ABB RobotStudio station: Task1_welding_1.rspag

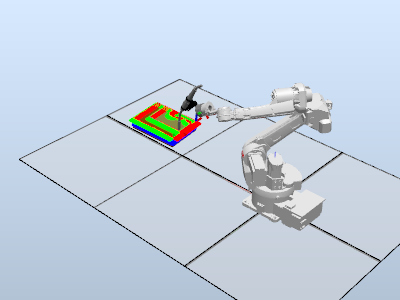
--- station ---
Station Task1_welding_1 (saved by RobotStudio 22.3.10098.0)
Controller IRB_1520ID_4kg_1.50m
  mechanical unit ROB_1: IRB1520ID_4_150__02, 6 joints, base frame (0, 0, 0) mm
Layout (positions relative to the parent item):
  - IRB1520ID_4_150__02 [mechanism, from Robots\IRB1520ID_4_150_G_02.rslib] at (0, 0, 0) mm; joint values [0.8708, -0.9702, 1.0298, -0.8942, 0.8494, 1.1291] (rad or m)
  - AW_Gun_PSF_25 [mechanism, from Tools\AW_Gun_PSF_25.rslib] at (433.02, 332.31, 841.28) mm, rotated rx 180 ry 59.43 rz -172.96 deg
  - Curve_thing [part, from Training Objects\Curve_Thing.rslib] at (696.55, 149.94, 458.64) mm, rotated rx 0 ry -5.23 rz 7.04 deg
  - Part_1 [part] at (696.55, 149.94, 458.64) mm, rotated rx 0 ry -5.23 rz 7.04 deg, size 300 x 200 x 0 mm
  - Part_2 [part] at (696.55, 149.94, 458.64) mm, rotated rx 0 ry -5.23 rz 7.04 deg, size 400 x 0 x 90 mm
Attachment: AW_Gun_PSF_25 is attached to IRB1520ID_4_150__02 / Link6

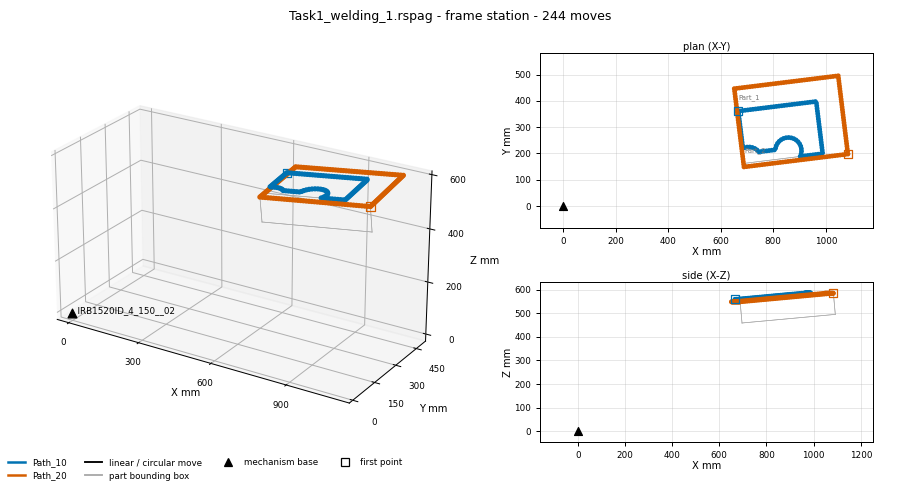
[picture p0: tool path of Task1_welding_1.rspag in frame station, 244 of 244 moves have a stored position in this frame; points joined in program order, loops and branches not executed]
--- Backups/IRB_1520ID_4kg_1.50m/RAPID/TASK1/PROGMOD/CalibData.mod ---
MODULE CalibData
	PERS tooldata AW_Gun:=[TRUE,[[119.5,0,352],[0.890213743,0,0.455543074,0]],[1,[0,0,100],[1,0,0,0],0,0,0]];
	TASK PERS wobjdata myPalletWO:=[FALSE,TRUE,"",[[688.418839009,148.925896983,548.269503166],[0.74843401,0.03415564,-0.030194721,-0.66164054]],[[0,0,0],[1,0,0,0]]];
    TASK PERS wobjdata Workobject_1:=[FALSE,TRUE,"",[[688.417832153,148.925979259,548.268984532],[0.997073299,0.002800799,-0.045502463,0.061371969]],[[0,0,0],[0,0.707106781,0.707106781,0]]];
    PROC Path_10()
        MoveJ Target_10,v1000,z100,AW_Gun\WObj:=wobj0;
        MoveL Target_20,v1000,z100,AW_Gun\WObj:=wobj0;
        MoveL Target_30,v1000,z100,AW_Gun\WObj:=wobj0;
        MoveL Target_40,v1000,z100,AW_Gun\WObj:=wobj0;
        MoveL Target_50,v1000,z100,AW_Gun\WObj:=wobj0;
        MoveL Target_60,v1000,z100,AW_Gun\WObj:=wobj0;
        MoveL Target_80,v1000,z100,AW_Gun\WObj:=wobj0;
        MoveL Target_70,v1000,z100,AW_Gun\WObj:=wobj0;
        MoveL Target_90,v1000,z100,AW_Gun\WObj:=wobj0;
        MoveL Target_100,v1000,z100,AW_Gun\WObj:=wobj0;
        MoveL Target_110,v1000,z100,AW_Gun\WObj:=wobj0;
        MoveL Target_120,v1000,z100,AW_Gun\WObj:=wobj0;
        MoveL Target_130,v1000,z100,AW_Gun\WObj:=wobj0;
        MoveL Target_140,v1000,z100,AW_Gun\WObj:=wobj0;
        MoveL Target_150,v1000,z100,AW_Gun\WObj:=wobj0;
        MoveL Target_160,v1000,z100,AW_Gun\WObj:=wobj0;
        MoveL Target_170,v1000,z100,AW_Gun\WObj:=wobj0;
        MoveL Target_180,v1000,z100,AW_Gun\WObj:=wobj0;
        MoveL Target_190,v1000,z100,AW_Gun\WObj:=wobj0;
        MoveL Target_200,v1000,z100,AW_Gun\WObj:=wobj0;
        MoveL Target_210,v1000,z100,AW_Gun\WObj:=wobj0;
        MoveL Target_220,v1000,z100,AW_Gun\WObj:=wobj0;
        MoveL Target_230,v1000,z100,AW_Gun\WObj:=wobj0;
        MoveL Target_240,v1000,z100,AW_Gun\WObj:=wobj0;
        MoveL Target_250,v1000,z100,AW_Gun\WObj:=wobj0;
        MoveL Target_260,v1000,z100,AW_Gun\WObj:=wobj0;
        MoveL Target_270,v1000,z100,AW_Gun\WObj:=wobj0;
        MoveL Target_280,v1000,z100,AW_Gun\WObj:=wobj0;
        MoveL Target_290,v1000,z100,AW_Gun\WObj:=wobj0;
        MoveL Target_300,v1000,z100,AW_Gun\WObj:=wobj0;
        MoveL Target_310,v1000,z100,AW_Gun\WObj:=wobj0;
        MoveL Target_320,v1000,z100,AW_Gun\WObj:=wobj0;
        MoveL Target_330,v1000,z100,AW_Gun\WObj:=wobj0;
        MoveL Target_340,v1000,z100,AW_Gun\WObj:=wobj0;
        MoveL Target_350,v1000,z100,AW_Gun\WObj:=wobj0;
        MoveL Target_360,v1000,z100,AW_Gun\WObj:=wobj0;
        MoveL Target_370,v1000,z100,AW_Gun\WObj:=wobj0;
        MoveL Target_380,v1000,z100,AW_Gun\WObj:=wobj0;
        MoveL Target_390,v1000,z100,AW_Gun\WObj:=wobj0;
        MoveL Target_400,v1000,z100,AW_Gun\WObj:=wobj0;
        MoveL Target_410,v1000,z100,AW_Gun\WObj:=wobj0;
        MoveL Target_420,v1000,z100,AW_Gun\WObj:=wobj0;
        MoveL Target_430,v1000,z100,AW_Gun\WObj:=wobj0;
        MoveL Target_440,v1000,z100,AW_Gun\WObj:=wobj0;
        MoveL Target_450,v1000,z100,AW_Gun\WObj:=wobj0;
        MoveL Target_460,v1000,z100,AW_Gun\WObj:=wobj0;
        MoveL Target_470,v1000,z100,AW_Gun\WObj:=wobj0;
        MoveL Target_480,v1000,z100,AW_Gun\WObj:=wobj0;
        MoveL Target_490,v1000,z100,AW_Gun\WObj:=wobj0;
        MoveL Target_500,v1000,z100,AW_Gun\WObj:=wobj0;
        MoveL Target_510,v1000,z100,AW_Gun\WObj:=wobj0;
        MoveL Target_520,v1000,z100,AW_Gun\WObj:=wobj0;
        MoveL Target_530,v1000,z100,AW_Gun\WObj:=wobj0;
        MoveL Target_540,v1000,z100,AW_Gun\WObj:=wobj0;
        MoveL Target_550,v1000,z100,AW_Gun\WObj:=wobj0;
        MoveL Target_560,v1000,z100,AW_Gun\WObj:=wobj0;
        MoveL Target_570,v1000,z100,AW_Gun\WObj:=wobj0;
        MoveL Target_580,v1000,z100,AW_Gun\WObj:=wobj0;
        MoveL Target_590,v1000,z100,AW_Gun\WObj:=wobj0;
        MoveL Target_600,v1000,z100,AW_Gun\WObj:=wobj0;
        MoveL Target_610,v1000,z100,AW_Gun\WObj:=wobj0;
        MoveL Target_620,v1000,z100,AW_Gun\WObj:=wobj0;
        MoveL Target_630,v1000,z100,AW_Gun\WObj:=wobj0;
        MoveL Target_640,v1000,z100,AW_Gun\WObj:=wobj0;
        MoveL Target_650,v1000,z100,AW_Gun\WObj:=wobj0;
        MoveL Target_660,v1000,z100,AW_Gun\WObj:=wobj0;
        MoveL Target_670,v1000,z100,AW_Gun\WObj:=wobj0;
        MoveL Target_680,v1000,z100,AW_Gun\WObj:=wobj0;
        MoveL Target_690,v1000,z100,AW_Gun\WObj:=wobj0;
        MoveL Target_700,v1000,z100,AW_Gun\WObj:=wobj0;
        MoveL Target_710,v1000,z100,AW_Gun\WObj:=wobj0;
        MoveL Target_720,v1000,z100,AW_Gun\WObj:=wobj0;
        MoveL Target_730,v1000,z100,AW_Gun\WObj:=wobj0;
        MoveL Target_740,v1000,z100,AW_Gun\WObj:=wobj0;
        MoveL Target_750,v1000,z100,AW_Gun\WObj:=wobj0;
        MoveL Target_760,v1000,z100,AW_Gun\WObj:=wobj0;
        MoveL Target_770,v1000,z100,AW_Gun\WObj:=wobj0;
        MoveL Target_780,v1000,z100,AW_Gun\WObj:=wobj0;
        MoveL Target_790,v1000,z100,AW_Gun\WObj:=wobj0;
        MoveL Target_800,v1000,z100,AW_Gun\WObj:=wobj0;
        MoveL Target_810,v1000,z100,AW_Gun\WObj:=wobj0;
        MoveL Target_820,v1000,z100,AW_Gun\WObj:=wobj0;
        MoveL Target_830,v1000,z100,AW_Gun\WObj:=wobj0;
        MoveL Target_840,v1000,z100,AW_Gun\WObj:=wobj0;
        MoveL Target_850,v1000,z100,AW_Gun\WObj:=wobj0;
        MoveL Target_860,v1000,z100,AW_Gun\WObj:=wobj0;
        MoveL Target_870,v1000,z100,AW_Gun\WObj:=wobj0;
        MoveL Target_880,v1000,z100,AW_Gun\WObj:=wobj0;
        MoveL Target_890,v1000,z100,AW_Gun\WObj:=wobj0;
        MoveL Target_900,v1000,z100,AW_Gun\WObj:=wobj0;
        MoveL Target_910,v1000,z100,AW_Gun\WObj:=wobj0;
        MoveL Target_920,v1000,z100,AW_Gun\WObj:=wobj0;
        MoveL Target_930,v1000,z100,AW_Gun\WObj:=wobj0;
        MoveL Target_940,v1000,z100,AW_Gun\WObj:=wobj0;
        MoveL Target_950,v1000,z100,AW_Gun\WObj:=wobj0;
        MoveL Target_960,v1000,z100,AW_Gun\WObj:=wobj0;
        MoveL Target_970,v1000,z100,AW_Gun\WObj:=wobj0;
        MoveL Target_980,v1000,z100,AW_Gun\WObj:=wobj0;
        MoveL Target_990,v1000,z100,AW_Gun\WObj:=wobj0;
        MoveL Target_1000,v1000,z100,AW_Gun\WObj:=wobj0;
        MoveL Target_1010,v1000,z100,AW_Gun\WObj:=wobj0;
        MoveL Target_1020,v1000,z100,AW_Gun\WObj:=wobj0;
        MoveL Target_1030,v1000,z100,AW_Gun\WObj:=wobj0;
        MoveL Target_1040,v1000,z100,AW_Gun\WObj:=wobj0;
    ENDPROC
    PROC Path_20()
        MoveJ Target_1050,v1000,z100,AW_Gun\WObj:=wobj0;
        MoveL Target_1060,v1000,z100,AW_Gun\WObj:=wobj0;
        MoveL Target_1070,v1000,z100,AW_Gun\WObj:=wobj0;
        MoveL Target_1080,v1000,z100,AW_Gun\WObj:=wobj0;
        MoveL Target_1090,v1000,z100,AW_Gun\WObj:=wobj0;
        MoveL Target_1100,v1000,z100,AW_Gun\WObj:=wobj0;
        MoveL Target_1110,v1000,z100,AW_Gun\WObj:=wobj0;
        MoveL Target_1120,v1000,z100,AW_Gun\WObj:=wobj0;
        MoveL Target_1130,v1000,z100,AW_Gun\WObj:=wobj0;
        MoveL Target_1140,v1000,z100,AW_Gun\WObj:=wobj0;
        MoveL Target_1150,v1000,z100,AW_Gun\WObj:=wobj0;
        MoveL Target_1160,v1000,z100,AW_Gun\WObj:=wobj0;
        MoveL Target_1170,v1000,z100,AW_Gun\WObj:=wobj0;
        MoveL Target_1180,v1000,z100,AW_Gun\WObj:=wobj0;
        MoveL Target_1190,v1000,z100,AW_Gun\WObj:=wobj0;
        MoveL Target_1200,v1000,z100,AW_Gun\WObj:=wobj0;
        MoveL Target_1210,v1000,z100,AW_Gun\WObj:=wobj0;
        MoveL Target_1220,v1000,z100,AW_Gun\WObj:=wobj0;
        MoveL Target_1230,v1000,z100,AW_Gun\WObj:=wobj0;
        MoveL Target_1240,v1000,z100,AW_Gun\WObj:=wobj0;
        MoveL Target_1250,v1000,z100,AW_Gun\WObj:=wobj0;
        MoveL Target_1260,v1000,z100,AW_Gun\WObj:=wobj0;
        MoveL Target_1270,v1000,z100,AW_Gun\WObj:=wobj0;
        MoveL Target_1280,v1000,z100,AW_Gun\WObj:=wobj0;
        MoveL Target_1290,v1000,z100,AW_Gun\WObj:=wobj0;
        MoveL Target_1300,v1000,z100,AW_Gun\WObj:=wobj0;
        MoveL Target_1310,v1000,z100,AW_Gun\WObj:=wobj0;
        MoveL Target_1320,v1000,z100,AW_Gun\WObj:=wobj0;
        MoveL Target_1330,v1000,z100,AW_Gun\WObj:=wobj0;
        MoveL Target_1340,v1000,z100,AW_Gun\WObj:=wobj0;
        MoveL Target_1350,v1000,z100,AW_Gun\WObj:=wobj0;
        MoveL Target_1360,v1000,z100,AW_Gun\WObj:=wobj0;
        MoveL Target_1370,v1000,z100,AW_Gun\WObj:=wobj0;
        MoveL Target_1380,v1000,z100,AW_Gun\WObj:=wobj0;
        MoveL Target_1390,v1000,z100,AW_Gun\WObj:=wobj0;
        MoveL Target_1400,v1000,z100,AW_Gun\WObj:=wobj0;
        MoveL Target_1410,v1000,z100,AW_Gun\WObj:=wobj0;
        MoveL Target_1420,v1000,z100,AW_Gun\WObj:=wobj0;
        MoveL Target_1430,v1000,z100,AW_Gun\WObj:=wobj0;
        MoveL Target_1440,v1000,z100,AW_Gun\WObj:=wobj0;
        MoveL Target_1450,v1000,z100,AW_Gun\WObj:=wobj0;
        MoveL Target_1460,v1000,z100,AW_Gun\WObj:=wobj0;
        MoveL Target_1470,v1000,z100,AW_Gun\WObj:=wobj0;
        MoveL Target_1480,v1000,z100,AW_Gun\WObj:=wobj0;
        MoveL Target_1490,v1000,z100,AW_Gun\WObj:=wobj0;
        MoveL Target_1500,v1000,z100,AW_Gun\WObj:=wobj0;
        MoveL Target_1510,v1000,z100,AW_Gun\WObj:=wobj0;
        MoveL Target_1520,v1000,z100,AW_Gun\WObj:=wobj0;
        MoveL Target_1530,v1000,z100,AW_Gun\WObj:=wobj0;
        MoveL Target_1540,v1000,z100,AW_Gun\WObj:=wobj0;
        MoveL Target_1550,v1000,z100,AW_Gun\WObj:=wobj0;
        MoveL Target_1560,v1000,z100,AW_Gun\WObj:=wobj0;
        MoveL Target_1570,v1000,z100,AW_Gun\WObj:=wobj0;
        MoveL Target_1580,v1000,z100,AW_Gun\WObj:=wobj0;
        MoveL Target_1590,v1000,z100,AW_Gun\WObj:=wobj0;
        MoveL Target_1600,v1000,z100,AW_Gun\WObj:=wobj0;
        MoveL Target_1610,v1000,z100,AW_Gun\WObj:=wobj0;
        MoveL Target_1620,v1000,z100,AW_Gun\WObj:=wobj0;
        MoveL Target_1630,v1000,z100,AW_Gun\WObj:=wobj0;
        MoveL Target_1640,v1000,z100,AW_Gun\WObj:=wobj0;
        MoveL Target_1650,v1000,z100,AW_Gun\WObj:=wobj0;
        MoveL Target_1660,v1000,z100,AW_Gun\WObj:=wobj0;
        MoveL Target_1670,v1000,z100,AW_Gun\WObj:=wobj0;
        MoveL Target_1680,v1000,z100,AW_Gun\WObj:=wobj0;
        MoveL Target_1690,v1000,z100,AW_Gun\WObj:=wobj0;
        MoveL Target_1700,v1000,z100,AW_Gun\WObj:=wobj0;
        MoveL Target_1710,v1000,z100,AW_Gun\WObj:=wobj0;
        MoveL Target_1720,v1000,z100,AW_Gun\WObj:=wobj0;
        MoveL Target_1730,v1000,z100,AW_Gun\WObj:=wobj0;
        MoveL Target_1740,v1000,z100,AW_Gun\WObj:=wobj0;
        MoveL Target_1750,v1000,z100,AW_Gun\WObj:=wobj0;
        MoveL Target_1760,v1000,z100,AW_Gun\WObj:=wobj0;
        MoveL Target_1770,v1000,z100,AW_Gun\WObj:=wobj0;
        MoveL Target_1780,v1000,z100,AW_Gun\WObj:=wobj0;
        MoveL Target_1790,v1000,z100,AW_Gun\WObj:=wobj0;
        MoveL Target_1800,v1000,z100,AW_Gun\WObj:=wobj0;
        MoveL Target_1810,v1000,z100,AW_Gun\WObj:=wobj0;
        MoveL Target_1820,v1000,z100,AW_Gun\WObj:=wobj0;
        MoveL Target_1830,v1000,z100,AW_Gun\WObj:=wobj0;
        MoveL Target_1840,v1000,z100,AW_Gun\WObj:=wobj0;
        MoveL Target_1850,v1000,z100,AW_Gun\WObj:=wobj0;
        MoveL Target_1860,v1000,z100,AW_Gun\WObj:=wobj0;
        MoveL Target_1870,v1000,z100,AW_Gun\WObj:=wobj0;
        MoveL Target_1880,v1000,z100,AW_Gun\WObj:=wobj0;
        MoveL Target_1890,v1000,z100,AW_Gun\WObj:=wobj0;
        MoveL Target_1900,v1000,z100,AW_Gun\WObj:=wobj0;
        MoveL Target_1910,v1000,z100,AW_Gun\WObj:=wobj0;
        MoveL Target_1920,v1000,z100,AW_Gun\WObj:=wobj0;
        MoveL Target_1930,v1000,z100,AW_Gun\WObj:=wobj0;
        MoveL Target_1940,v1000,z100,AW_Gun\WObj:=wobj0;
        MoveL Target_1950,v1000,z100,AW_Gun\WObj:=wobj0;
        MoveL Target_1960,v1000,z100,AW_Gun\WObj:=wobj0;
        MoveL Target_1970,v1000,z100,AW_Gun\WObj:=wobj0;
        MoveL Target_1980,v1000,z100,AW_Gun\WObj:=wobj0;
        MoveL Target_1990,v1000,z100,AW_Gun\WObj:=wobj0;
        MoveL Target_2000,v1000,z100,AW_Gun\WObj:=wobj0;
        MoveL Target_2010,v1000,z100,AW_Gun\WObj:=wobj0;
        MoveL Target_2020,v1000,z100,AW_Gun\WObj:=wobj0;
        MoveL Target_2030,v1000,z100,AW_Gun\WObj:=wobj0;
        MoveL Target_2040,v1000,z100,AW_Gun\WObj:=wobj0;
        MoveL Target_2050,v1000,z100,AW_Gun\WObj:=wobj0;
        MoveL Target_2060,v1000,z100,AW_Gun\WObj:=wobj0;
        MoveL Target_2070,v1000,z100,AW_Gun\WObj:=wobj0;
        MoveL Target_2080,v1000,z100,AW_Gun\WObj:=wobj0;
        MoveL Target_2090,v1000,z100,AW_Gun\WObj:=wobj0;
        MoveL Target_2100,v1000,z100,AW_Gun\WObj:=wobj0;
        MoveL Target_2110,v1000,z100,AW_Gun\WObj:=wobj0;
        MoveL Target_2120,v1000,z100,AW_Gun\WObj:=wobj0;
        MoveL Target_2130,v1000,z100,AW_Gun\WObj:=wobj0;
        MoveL Target_2140,v1000,z100,AW_Gun\WObj:=wobj0;
        MoveL Target_2150,v1000,z100,AW_Gun\WObj:=wobj0;
        MoveL Target_2160,v1000,z100,AW_Gun\WObj:=wobj0;
        MoveL Target_2170,v1000,z100,AW_Gun\WObj:=wobj0;
        MoveL Target_2180,v1000,z100,AW_Gun\WObj:=wobj0;
        MoveL Target_2190,v1000,z100,AW_Gun\WObj:=wobj0;
        MoveL Target_2200,v1000,z100,AW_Gun\WObj:=wobj0;
        MoveL Target_2210,v1000,z100,AW_Gun\WObj:=wobj0;
        MoveL Target_2220,v1000,z100,AW_Gun\WObj:=wobj0;
        MoveL Target_2230,v1000,z100,AW_Gun\WObj:=wobj0;
        MoveL Target_2240,v1000,z100,AW_Gun\WObj:=wobj0;
        MoveL Target_2250,v1000,z100,AW_Gun\WObj:=wobj0;
        MoveL Target_2260,v1000,z100,AW_Gun\WObj:=wobj0;
        MoveL Target_2270,v1000,z100,AW_Gun\WObj:=wobj0;
        MoveL Target_2280,v1000,z100,AW_Gun\WObj:=wobj0;
        MoveL Target_2290,v1000,z100,AW_Gun\WObj:=wobj0;
        MoveL Target_2300,v1000,z100,AW_Gun\WObj:=wobj0;
        MoveL Target_2310,v1000,z100,AW_Gun\WObj:=wobj0;
        MoveL Target_2320,v1000,z100,AW_Gun\WObj:=wobj0;
        MoveL Target_2330,v1000,z100,AW_Gun\WObj:=wobj0;
        MoveL Target_2340,v1000,z100,AW_Gun\WObj:=wobj0;
        MoveL Target_2350,v1000,z100,AW_Gun\WObj:=wobj0;
        MoveL Target_2360,v1000,z100,AW_Gun\WObj:=wobj0;
        MoveL Target_2370,v1000,z100,AW_Gun\WObj:=wobj0;
        MoveL Target_2380,v1000,z100,AW_Gun\WObj:=wobj0;
        MoveL Target_2390,v1000,z100,AW_Gun\WObj:=wobj0;
        MoveL Target_2400,v1000,z100,AW_Gun\WObj:=wobj0;
        MoveL Target_2410,v1000,z100,AW_Gun\WObj:=wobj0;
        MoveL Target_2420,v1000,z100,AW_Gun\WObj:=wobj0;
        MoveL Target_2430,v1000,z100,AW_Gun\WObj:=wobj0;
        MoveL Target_2440,v1000,z100,AW_Gun\WObj:=wobj0;
    ENDPROC
ENDMODULE

--- Backups/IRB_1520ID_4kg_1.50m/RAPID/TASK1/PROGMOD/Module1.mod ---
MODULE Module1


        CONST robtarget Target_10:=[[666.736269094,361.19507219,558.723843353],[0.045502886,-0.061372268,0.997073261,0.002800813],[0,0,0,0],[9E+09,9E+09,9E+09,9E+09,9E+09,9E+09]];
    CONST robtarget Target_20:=[[667.962670945,351.270560187,558.723843353],[0.045502886,-0.061372268,0.997073261,0.002800813],[0,0,0,0],[9E+09,9E+09,9E+09,9E+09,9E+09,9E+09]];
    CONST robtarget Target_30:=[[669.189072796,341.346048184,558.723843353],[0.045502886,-0.061372268,0.997073261,0.002800813],[0,0,0,0],[9E+09,9E+09,9E+09,9E+09,9E+09,9E+09]];
    CONST robtarget Target_40:=[[670.415474647,331.421536181,558.723843353],[0.045502886,-0.061372268,0.997073261,0.002800813],[0,0,0,0],[9E+09,9E+09,9E+09,9E+09,9E+09,9E+09]];
    CONST robtarget Target_50:=[[671.641876498,321.497024178,558.723843353],[0.045502886,-0.061372268,0.997073261,0.002800813],[0,0,0,0],[9E+09,9E+09,9E+09,9E+09,9E+09,9E+09]];
    CONST robtarget Target_60:=[[672.868278349,311.572512174,558.723843353],[0.045502886,-0.061372268,0.997073261,0.002800813],[0,0,0,0],[9E+09,9E+09,9E+09,9E+09,9E+09,9E+09]];
    CONST robtarget Target_70:=[[674.0946802,301.648000171,558.723843353],[0.045502886,-0.061372268,0.997073261,0.002800813],[0,0,0,0],[9E+09,9E+09,9E+09,9E+09,9E+09,9E+09]];
    CONST robtarget Target_80:=[[675.321082051,291.723488168,558.723843353],[0.045502886,-0.061372268,0.997073261,0.002800813],[0,0,0,0],[9E+09,9E+09,9E+09,9E+09,9E+09,9E+09]];
    CONST robtarget Target_90:=[[676.547483902,281.798976165,558.723843353],[0.045502886,-0.061372268,0.997073261,0.002800813],[0,0,0,0],[9E+09,9E+09,9E+09,9E+09,9E+09,9E+09]];
    CONST robtarget Target_100:=[[677.773885753,271.874464162,558.723843353],[0.045502886,-0.061372268,0.997073261,0.002800813],[0,0,0,0],[9E+09,9E+09,9E+09,9E+09,9E+09,9E+09]];
    CONST robtarget Target_110:=[[679.000287604,261.949952159,558.723843353],[0.045502886,-0.061372268,0.997073261,0.002800813],[0,0,0,0],[9E+09,9E+09,9E+09,9E+09,9E+09,9E+09]];
    CONST robtarget Target_120:=[[680.226689455,252.025440156,558.723843353],[0.045502886,-0.061372268,0.997073261,0.002800813],[0,0,0,0],[9E+09,9E+09,9E+09,9E+09,9E+09,9E+09]];
    CONST robtarget Target_130:=[[681.453091306,242.100928153,558.723843353],[0.045502886,-0.061372268,0.997073261,0.002800813],[0,0,0,0],[9E+09,9E+09,9E+09,9E+09,9E+09,9E+09]];
    CONST robtarget Target_140:=[[682.679493157,232.17641615,558.723843353],[0.045502886,-0.061372268,0.997073261,0.002800813],[0,0,0,0],[9E+09,9E+09,9E+09,9E+09,9E+09,9E+09]];
    CONST robtarget Target_150:=[[683.905895008,222.251904146,558.723843353],[0.045502886,-0.061372268,0.997073261,0.002800813],[0,0,0,0],[9E+09,9E+09,9E+09,9E+09,9E+09,9E+09]];
    CONST robtarget Target_160:=[[690.804802544,222.13014152,559.348711753],[0.045502886,-0.061372268,0.997073261,0.002800813],[0,0,0,0],[9E+09,9E+09,9E+09,9E+09,9E+09,9E+09]];
    CONST robtarget Target_170:=[[700.500489926,224.330621813,560.253500924],[0.045502886,-0.061372268,0.997073261,0.002800813],[0,0,0,0],[9E+09,9E+09,9E+09,9E+09,9E+09,9E+09]];
    CONST robtarget Target_180:=[[710.440267778,224.552761127,561.158255685],[0.045502886,-0.061372268,0.997073261,0.002800813],[0,0,0,0],[9E+09,9E+09,9E+09,9E+09,9E+09,9E+09]];
    CONST robtarget Target_190:=[[720.227868523,222.787703468,562.026906317],[0.045502886,-0.061372268,0.997073261,0.002800813],[0,0,0,0],[9E+09,9E+09,9E+09,9E+09,9E+09,9E+09]];
    CONST robtarget Target_200:=[[729.473091405,219.105816114,562.824822462],[0.045502886,-0.061372268,0.997073261,0.002800813],[0,0,0,0],[9E+09,9E+09,9E+09,9E+09,9E+09,9E+09]];
    CONST robtarget Target_210:=[[737.807358563,213.653884297,563.520193721],[0.045502886,-0.061372268,0.997073261,0.002800813],[0,0,0,0],[9E+09,9E+09,9E+09,9E+09,9E+09,9E+09]];
    CONST robtarget Target_220:=[[744.898409066,206.649259332,564.085297836],[0.045502886,-0.061372268,0.997073261,0.002800813],[0,0,0,0],[9E+09,9E+09,9E+09,9E+09,9E+09,9E+09]];
    CONST robtarget Target_230:=[[754.627167172,207.480999334,564.977735655],[0.045502886,-0.061372268,0.997073261,0.002800813],[0,0,0,0],[9E+09,9E+09,9E+09,9E+09,9E+09,9E+09]];
    CONST robtarget Target_240:=[[764.510425813,208.702303383,565.888567718],[0.045502886,-0.061372268,0.997073261,0.002800813],[0,0,0,0],[9E+09,9E+09,9E+09,9E+09,9E+09,9E+09]];
    CONST robtarget Target_250:=[[774.393684454,209.923607432,566.799399781],[0.045502886,-0.061372268,0.997073261,0.002800813],[0,0,0,0],[9E+09,9E+09,9E+09,9E+09,9E+09,9E+09]];
    CONST robtarget Target_260:=[[784.276943096,211.14491148,567.710231845],[0.045502886,-0.061372268,0.997073261,0.002800813],[0,0,0,0],[9E+09,9E+09,9E+09,9E+09,9E+09,9E+09]];
    CONST robtarget Target_270:=[[794.160201737,212.366215529,568.621063908],[0.045502886,-0.061372268,0.997073261,0.002800813],[0,0,0,0],[9E+09,9E+09,9E+09,9E+09,9E+09,9E+09]];
    CONST robtarget Target_280:=[[804.043460379,213.587519578,569.531895971],[0.045502886,-0.061372268,0.997073261,0.002800813],[0,0,0,0],[9E+09,9E+09,9E+09,9E+09,9E+09,9E+09]];
    CONST robtarget Target_290:=[[808.628332921,220.148142904,570.021669484],[0.045502886,-0.061372268,0.997073261,0.002800813],[0,0,0,0],[9E+09,9E+09,9E+09,9E+09,9E+09,9E+09]];
    CONST robtarget Target_300:=[[811.455727345,229.7158216,570.38564192],[0.045502886,-0.061372268,0.997073261,0.002800813],[0,0,0,0],[9E+09,9E+09,9E+09,9E+09,9E+09,9E+09]];
    CONST robtarget Target_310:=[[816.120473083,238.526865532,570.907908924],[0.045502886,-0.061372268,0.997073261,0.002800813],[0,0,0,0],[9E+09,9E+09,9E+09,9E+09,9E+09,9E+09]];
    CONST robtarget Target_320:=[[822.436601444,246.230006182,571.56764936],[0.045502886,-0.061372268,0.997073261,0.002800813],[0,0,0,0],[9E+09,9E+09,9E+09,9E+09,9E+09,9E+09]];
    CONST robtarget Target_330:=[[830.152308321,252.518143643,572.338561459],[0.045502886,-0.061372268,0.997073261,0.002800813],[0,0,0,0],[9E+09,9E+09,9E+09,9E+09,9E+09,9E+09]];
    CONST robtarget Target_340:=[[838.959992829,257.140589716,573.189911388],[0.045502886,-0.061372268,0.997073261,0.002800813],[0,0,0,0],[9E+09,9E+09,9E+09,9E+09,9E+09,9E+09]];
    CONST robtarget Target_350:=[[848.508520381,259.913062063,574.087758512],[0.045502886,-0.061372268,0.997073261,0.002800813],[0,0,0,0],[9E+09,9E+09,9E+09,9E+09,9E+09,9E+09]];
    CONST robtarget Target_360:=[[858.417221316,260.725030962,574.996308499],[0.045502886,-0.061372268,0.997073261,0.002800813],[0,0,0,0],[9E+09,9E+09,9E+09,9E+09,9E+09,9E+09]];
    CONST robtarget Target_370:=[[868.291066997,259.544125775,575.879340329],[0.045502886,-0.061372268,0.997073261,0.002800813],[0,0,0,0],[9E+09,9E+09,9E+09,9E+09,9E+09,9E+09]];
    CONST robtarget Target_380:=[[877.736418354,256.417425464,576.701650308],[0.045502886,-0.061372268,0.997073261,0.002800813],[0,0,0,0],[9E+09,9E+09,9E+09,9E+09,9E+09,9E+09]];
    CONST robtarget Target_390:=[[886.376719035,251.469581705,577.430455534],[0.045502886,-0.061372268,0.997073261,0.002800813],[0,0,0,0],[9E+09,9E+09,9E+09,9E+09,9E+09,9E+09]];
    CONST robtarget Target_400:=[[893.86750752,244.897849414,578.036700841],[0.045502886,-0.061372268,0.997073261,0.002800813],[0,0,0,0],[9E+09,9E+09,9E+09,9E+09,9E+09,9E+09]];
    CONST robtarget Target_410:=[[899.910149708,236.964222819,578.496217143],[0.045502886,-0.061372268,0.997073261,0.002800813],[0,0,0,0],[9E+09,9E+09,9E+09,9E+09,9E+09,9E+09]];
    CONST robtarget Target_420:=[[904.263744525,227.984990577,578.790684974],[0.045502886,-0.061372268,0.997073261,0.002800813],[0,0,0,0],[9E+09,9E+09,9E+09,9E+09,9E+09,9E+09]];
    CONST robtarget Target_430:=[[906.754727884,218.318126341,578.908364832],[0.045502886,-0.061372268,0.997073261,0.002800813],[0,0,0,0],[9E+09,9E+09,9E+09,9E+09,9E+09,9E+09]];
    CONST robtarget Target_440:=[[907.283792139,208.349017484,578.844565191],[0.045502886,-0.061372268,0.997073261,0.002800813],[0,0,0,0],[9E+09,9E+09,9E+09,9E+09,9E+09,9E+09]];
    CONST robtarget Target_450:=[[905.829845169,198.475100915,578.601829542],[0.045502886,-0.061372268,0.997073261,0.002800813],[0,0,0,0],[9E+09,9E+09,9E+09,9E+09,9E+09,9E+09]];
    CONST robtarget Target_460:=[[902.450851249,189.09001853,578.18983499],[0.045502886,-0.061372268,0.997073261,0.002800813],[0,0,0,0],[9E+09,9E+09,9E+09,9E+09,9E+09,9E+09]];
    CONST robtarget Target_470:=[[911.849942658,189.963263864,579.052813558],[0.045502886,-0.061372268,0.997073261,0.002800813],[0,0,0,0],[9E+09,9E+09,9E+09,9E+09,9E+09,9E+09]];
    CONST robtarget Target_480:=[[921.733201299,191.184567913,579.963645621],[0.045502886,-0.061372268,0.997073261,0.002800813],[0,0,0,0],[9E+09,9E+09,9E+09,9E+09,9E+09,9E+09]];
    CONST robtarget Target_490:=[[931.616459941,192.405871962,580.874477684],[0.045502886,-0.061372268,0.997073261,0.002800813],[0,0,0,0],[9E+09,9E+09,9E+09,9E+09,9E+09,9E+09]];
    CONST robtarget Target_500:=[[941.499718582,193.627176011,581.785309747],[0.045502886,-0.061372268,0.997073261,0.002800813],[0,0,0,0],[9E+09,9E+09,9E+09,9E+09,9E+09,9E+09]];
    CONST robtarget Target_510:=[[951.382977224,194.84848006,582.696141811],[0.045502886,-0.061372268,0.997073261,0.002800813],[0,0,0,0],[9E+09,9E+09,9E+09,9E+09,9E+09,9E+09]];
    CONST robtarget Target_520:=[[961.266235865,196.069784108,583.606973874],[0.045502886,-0.061372268,0.997073261,0.002800813],[0,0,0,0],[9E+09,9E+09,9E+09,9E+09,9E+09,9E+09]];
    CONST robtarget Target_530:=[[971.149494506,197.291088157,584.517805937],[0.045502886,-0.061372268,0.997073261,0.002800813],[0,0,0,0],[9E+09,9E+09,9E+09,9E+09,9E+09,9E+09]];
    CONST robtarget Target_540:=[[981.032753148,198.512392206,585.428638],[0.045502886,-0.061372268,0.997073261,0.002800813],[0,0,0,0],[9E+09,9E+09,9E+09,9E+09,9E+09,9E+09]];
    CONST robtarget Target_550:=[[987.370695882,202.511064801,586.048805249],[0.045502886,-0.061372268,0.997073261,0.002800813],[0,0,0,0],[9E+09,9E+09,9E+09,9E+09,9E+09,9E+09]];
    CONST robtarget Target_560:=[[986.144294031,212.435576804,586.048805249],[0.045502886,-0.061372268,0.997073261,0.002800813],[0,0,0,0],[9E+09,9E+09,9E+09,9E+09,9E+09,9E+09]];
    CONST robtarget Target_570:=[[984.91789218,222.360088807,586.048805249],[0.045502886,-0.061372268,0.997073261,0.002800813],[0,0,0,0],[9E+09,9E+09,9E+09,9E+09,9E+09,9E+09]];
    CONST robtarget Target_580:=[[983.691490329,232.28460081,586.048805249],[0.045502886,-0.061372268,0.997073261,0.002800813],[0,0,0,0],[9E+09,9E+09,9E+09,9E+09,9E+09,9E+09]];
    CONST robtarget Target_590:=[[982.465088478,242.209112813,586.048805249],[0.045502886,-0.061372268,0.997073261,0.002800813],[0,0,0,0],[9E+09,9E+09,9E+09,9E+09,9E+09,9E+09]];
    CONST robtarget Target_600:=[[981.238686627,252.133624816,586.048805249],[0.045502886,-0.061372268,0.997073261,0.002800813],[0,0,0,0],[9E+09,9E+09,9E+09,9E+09,9E+09,9E+09]];
    CONST robtarget Target_610:=[[980.012284776,262.058136819,586.048805249],[0.045502886,-0.061372268,0.997073261,0.002800813],[0,0,0,0],[9E+09,9E+09,9E+09,9E+09,9E+09,9E+09]];
    CONST robtarget Target_620:=[[978.785882925,271.982648822,586.048805249],[0.045502886,-0.061372268,0.997073261,0.002800813],[0,0,0,0],[9E+09,9E+09,9E+09,9E+09,9E+09,9E+09]];
    CONST robtarget Target_630:=[[977.559481074,281.907160826,586.048805249],[0.045502886,-0.061372268,0.997073261,0.002800813],[0,0,0,0],[9E+09,9E+09,9E+09,9E+09,9E+09,9E+09]];
    CONST robtarget Target_640:=[[976.333079223,291.831672829,586.048805249],[0.045502886,-0.061372268,0.997073261,0.002800813],[0,0,0,0],[9E+09,9E+09,9E+09,9E+09,9E+09,9E+09]];
    CONST robtarget Target_650:=[[975.106677372,301.756184832,586.048805249],[0.045502886,-0.061372268,0.997073261,0.002800813],[0,0,0,0],[9E+09,9E+09,9E+09,9E+09,9E+09,9E+09]];
    CONST robtarget Target_660:=[[973.880275521,311.680696835,586.048805249],[0.045502886,-0.061372268,0.997073261,0.002800813],[0,0,0,0],[9E+09,9E+09,9E+09,9E+09,9E+09,9E+09]];
    CONST robtarget Target_670:=[[972.65387367,321.605208838,586.048805249],[0.045502886,-0.061372268,0.997073261,0.002800813],[0,0,0,0],[9E+09,9E+09,9E+09,9E+09,9E+09,9E+09]];
    CONST robtarget Target_680:=[[971.427471819,331.529720841,586.048805249],[0.045502886,-0.061372268,0.997073261,0.002800813],[0,0,0,0],[9E+09,9E+09,9E+09,9E+09,9E+09,9E+09]];
    CONST robtarget Target_690:=[[970.201069968,341.454232844,586.048805249],[0.045502886,-0.061372268,0.997073261,0.002800813],[0,0,0,0],[9E+09,9E+09,9E+09,9E+09,9E+09,9E+09]];
    CONST robtarget Target_700:=[[968.974668117,351.378744847,586.048805249],[0.045502886,-0.061372268,0.997073261,0.002800813],[0,0,0,0],[9E+09,9E+09,9E+09,9E+09,9E+09,9E+09]];
    CONST robtarget Target_710:=[[967.748266266,361.30325685,586.048805249],[0.045502886,-0.061372268,0.997073261,0.002800813],[0,0,0,0],[9E+09,9E+09,9E+09,9E+09,9E+09,9E+09]];
    CONST robtarget Target_720:=[[966.521864415,371.227768854,586.048805249],[0.045502886,-0.061372268,0.997073261,0.002800813],[0,0,0,0],[9E+09,9E+09,9E+09,9E+09,9E+09,9E+09]];
    CONST robtarget Target_730:=[[965.295462564,381.152280857,586.048805249],[0.045502886,-0.061372268,0.997073261,0.002800813],[0,0,0,0],[9E+09,9E+09,9E+09,9E+09,9E+09,9E+09]];
    CONST robtarget Target_740:=[[964.069060713,391.07679286,586.048805249],[0.045502886,-0.061372268,0.997073261,0.002800813],[0,0,0,0],[9E+09,9E+09,9E+09,9E+09,9E+09,9E+09]];
    CONST robtarget Target_750:=[[960.080081904,397.44445099,585.758140435],[0.045502886,-0.061372268,0.997073261,0.002800813],[0,0,0,0],[9E+09,9E+09,9E+09,9E+09,9E+09,9E+09]];
    CONST robtarget Target_760:=[[950.196823262,396.223146941,584.847308372],[0.045502886,-0.061372268,0.997073261,0.002800813],[0,0,0,0],[9E+09,9E+09,9E+09,9E+09,9E+09,9E+09]];
    CONST robtarget Target_770:=[[940.313564621,395.001842892,583.936476309],[0.045502886,-0.061372268,0.997073261,0.002800813],[0,0,0,0],[9E+09,9E+09,9E+09,9E+09,9E+09,9E+09]];
    CONST robtarget Target_780:=[[930.430305979,393.780538843,583.025644245],[0.045502886,-0.061372268,0.997073261,0.002800813],[0,0,0,0],[9E+09,9E+09,9E+09,9E+09,9E+09,9E+09]];
    CONST robtarget Target_790:=[[920.547047338,392.559234795,582.114812182],[0.045502886,-0.061372268,0.997073261,0.002800813],[0,0,0,0],[9E+09,9E+09,9E+09,9E+09,9E+09,9E+09]];
    CONST robtarget Target_800:=[[910.663788697,391.337930746,581.203980119],[0.045502886,-0.061372268,0.997073261,0.002800813],[0,0,0,0],[9E+09,9E+09,9E+09,9E+09,9E+09,9E+09]];
    CONST robtarget Target_810:=[[900.780530055,390.116626697,580.293148056],[0.045502886,-0.061372268,0.997073261,0.002800813],[0,0,0,0],[9E+09,9E+09,9E+09,9E+09,9E+09,9E+09]];
    CONST robtarget Target_820:=[[890.897271414,388.895322648,579.382315993],[0.045502886,-0.061372268,0.997073261,0.002800813],[0,0,0,0],[9E+09,9E+09,9E+09,9E+09,9E+09,9E+09]];
    CONST robtarget Target_830:=[[881.014012772,387.674018599,578.471483929],[0.045502886,-0.061372268,0.997073261,0.002800813],[0,0,0,0],[9E+09,9E+09,9E+09,9E+09,9E+09,9E+09]];
    CONST robtarget Target_840:=[[871.130754131,386.452714551,577.560651866],[0.045502886,-0.061372268,0.997073261,0.002800813],[0,0,0,0],[9E+09,9E+09,9E+09,9E+09,9E+09,9E+09]];
    CONST robtarget Target_850:=[[861.24749549,385.231410502,576.649819803],[0.045502886,-0.061372268,0.997073261,0.002800813],[0,0,0,0],[9E+09,9E+09,9E+09,9E+09,9E+09,9E+09]];
    CONST robtarget Target_860:=[[851.364236848,384.010106453,575.73898774],[0.045502886,-0.061372268,0.997073261,0.002800813],[0,0,0,0],[9E+09,9E+09,9E+09,9E+09,9E+09,9E+09]];
    CONST robtarget Target_870:=[[841.480978207,382.788802404,574.828155677],[0.045502886,-0.061372268,0.997073261,0.002800813],[0,0,0,0],[9E+09,9E+09,9E+09,9E+09,9E+09,9E+09]];
    CONST robtarget Target_880:=[[831.597719565,381.567498356,573.917323614],[0.045502886,-0.061372268,0.997073261,0.002800813],[0,0,0,0],[9E+09,9E+09,9E+09,9E+09,9E+09,9E+09]];
    CONST robtarget Target_890:=[[821.714460924,380.346194307,573.00649155],[0.045502886,-0.061372268,0.997073261,0.002800813],[0,0,0,0],[9E+09,9E+09,9E+09,9E+09,9E+09,9E+09]];
    CONST robtarget Target_900:=[[811.831202282,379.124890258,572.095659487],[0.045502886,-0.061372268,0.997073261,0.002800813],[0,0,0,0],[9E+09,9E+09,9E+09,9E+09,9E+09,9E+09]];
    CONST robtarget Target_910:=[[801.947943641,377.903586209,571.184827424],[0.045502886,-0.061372268,0.997073261,0.002800813],[0,0,0,0],[9E+09,9E+09,9E+09,9E+09,9E+09,9E+09]];
    CONST robtarget Target_920:=[[792.064685,376.68228216,570.273995361],[0.045502886,-0.061372268,0.997073261,0.002800813],[0,0,0,0],[9E+09,9E+09,9E+09,9E+09,9E+09,9E+09]];
    CONST robtarget Target_930:=[[782.181426358,375.460978112,569.363163298],[0.045502886,-0.061372268,0.997073261,0.002800813],[0,0,0,0],[9E+09,9E+09,9E+09,9E+09,9E+09,9E+09]];
    CONST robtarget Target_940:=[[772.298167717,374.239674063,568.452331234],[0.045502886,-0.061372268,0.997073261,0.002800813],[0,0,0,0],[9E+09,9E+09,9E+09,9E+09,9E+09,9E+09]];
    CONST robtarget Target_950:=[[762.414909075,373.018370014,567.541499171],[0.045502886,-0.061372268,0.997073261,0.002800813],[0,0,0,0],[9E+09,9E+09,9E+09,9E+09,9E+09,9E+09]];
    CONST robtarget Target_960:=[[752.531650434,371.797065965,566.630667108],[0.045502886,-0.061372268,0.997073261,0.002800813],[0,0,0,0],[9E+09,9E+09,9E+09,9E+09,9E+09,9E+09]];
    CONST robtarget Target_970:=[[742.648391793,370.575761917,565.719835045],[0.045502886,-0.061372268,0.997073261,0.002800813],[0,0,0,0],[9E+09,9E+09,9E+09,9E+09,9E+09,9E+09]];
    CONST robtarget Target_980:=[[732.765133151,369.354457868,564.809002982],[0.045502886,-0.061372268,0.997073261,0.002800813],[0,0,0,0],[9E+09,9E+09,9E+09,9E+09,9E+09,9E+09]];
    CONST robtarget Target_990:=[[722.88187451,368.133153819,563.898170918],[0.045502886,-0.061372268,0.997073261,0.002800813],[0,0,0,0],[9E+09,9E+09,9E+09,9E+09,9E+09,9E+09]];
    CONST robtarget Target_1000:=[[712.998615868,366.91184977,562.987338855],[0.045502886,-0.061372268,0.997073261,0.002800813],[0,0,0,0],[9E+09,9E+09,9E+09,9E+09,9E+09,9E+09]];
    CONST robtarget Target_1010:=[[703.115357227,365.690545721,562.076506792],[0.045502886,-0.061372268,0.997073261,0.002800813],[0,0,0,0],[9E+09,9E+09,9E+09,9E+09,9E+09,9E+09]];
    CONST robtarget Target_1020:=[[693.232098586,364.469241673,561.165674729],[0.045502886,-0.061372268,0.997073261,0.002800813],[0,0,0,0],[9E+09,9E+09,9E+09,9E+09,9E+09,9E+09]];
    CONST robtarget Target_1030:=[[683.348839944,363.247937624,560.254842666],[0.045502886,-0.061372268,0.997073261,0.002800813],[0,0,0,0],[9E+09,9E+09,9E+09,9E+09,9E+09,9E+09]];
    CONST robtarget Target_1040:=[[673.465581303,362.026633575,559.344010602],[0.045502886,-0.061372268,0.997073261,0.002800813],[0,0,0,0],[9E+09,9E+09,9E+09,9E+09,9E+09,9E+09]];
    CONST robtarget Target_1050:=[[1083.748761163,197.777785165,584.702492742],[0.045502886,-0.061372268,0.997073261,0.002800813],[0,0,0,0],[9E+09,9E+09,9E+09,9E+09,9E+09,9E+09]];
    CONST robtarget Target_1060:=[[1082.522359312,207.702297168,584.702492742],[0.045502886,-0.061372268,0.997073261,0.002800813],[0,0,0,0],[9E+09,9E+09,9E+09,9E+09,9E+09,9E+09]];
    CONST robtarget Target_1070:=[[1081.295957461,217.626809171,584.702492742],[0.045502886,-0.061372268,0.997073261,0.002800813],[0,0,0,0],[9E+09,9E+09,9E+09,9E+09,9E+09,9E+09]];
    CONST robtarget Target_1080:=[[1080.06955561,227.551321174,584.702492742],[0.045502886,-0.061372268,0.997073261,0.002800813],[0,0,0,0],[9E+09,9E+09,9E+09,9E+09,9E+09,9E+09]];
    CONST robtarget Target_1090:=[[1078.843153759,237.475833177,584.702492742],[0.045502886,-0.061372268,0.997073261,0.002800813],[0,0,0,0],[9E+09,9E+09,9E+09,9E+09,9E+09,9E+09]];
    CONST robtarget Target_1100:=[[1077.616751908,247.400345181,584.702492742],[0.045502886,-0.061372268,0.997073261,0.002800813],[0,0,0,0],[9E+09,9E+09,9E+09,9E+09,9E+09,9E+09]];
    CONST robtarget Target_1110:=[[1076.390350057,257.324857184,584.702492742],[0.045502886,-0.061372268,0.997073261,0.002800813],[0,0,0,0],[9E+09,9E+09,9E+09,9E+09,9E+09,9E+09]];
    CONST robtarget Target_1120:=[[1075.163948206,267.249369187,584.702492742],[0.045502886,-0.061372268,0.997073261,0.002800813],[0,0,0,0],[9E+09,9E+09,9E+09,9E+09,9E+09,9E+09]];
    CONST robtarget Target_1130:=[[1073.937546355,277.17388119,584.702492742],[0.045502886,-0.061372268,0.997073261,0.002800813],[0,0,0,0],[9E+09,9E+09,9E+09,9E+09,9E+09,9E+09]];
    CONST robtarget Target_1140:=[[1072.711144504,287.098393193,584.702492742],[0.045502886,-0.061372268,0.997073261,0.002800813],[0,0,0,0],[9E+09,9E+09,9E+09,9E+09,9E+09,9E+09]];
    CONST robtarget Target_1150:=[[1071.484742653,297.022905196,584.702492742],[0.045502886,-0.061372268,0.997073261,0.002800813],[0,0,0,0],[9E+09,9E+09,9E+09,9E+09,9E+09,9E+09]];
    CONST robtarget Target_1160:=[[1070.258340802,306.947417199,584.702492742],[0.045502886,-0.061372268,0.997073261,0.002800813],[0,0,0,0],[9E+09,9E+09,9E+09,9E+09,9E+09,9E+09]];
    CONST robtarget Target_1170:=[[1069.031938951,316.871929202,584.702492742],[0.045502886,-0.061372268,0.997073261,0.002800813],[0,0,0,0],[9E+09,9E+09,9E+09,9E+09,9E+09,9E+09]];
    CONST robtarget Target_1180:=[[1067.8055371,326.796441205,584.702492742],[0.045502886,-0.061372268,0.997073261,0.002800813],[0,0,0,0],[9E+09,9E+09,9E+09,9E+09,9E+09,9E+09]];
    CONST robtarget Target_1190:=[[1066.579135249,336.720953209,584.702492742],[0.045502886,-0.061372268,0.997073261,0.002800813],[0,0,0,0],[9E+09,9E+09,9E+09,9E+09,9E+09,9E+09]];
    CONST robtarget Target_1200:=[[1065.352733398,346.645465212,584.702492742],[0.045502886,-0.061372268,0.997073261,0.002800813],[0,0,0,0],[9E+09,9E+09,9E+09,9E+09,9E+09,9E+09]];
    CONST robtarget Target_1210:=[[1064.126331547,356.569977215,584.702492742],[0.045502886,-0.061372268,0.997073261,0.002800813],[0,0,0,0],[9E+09,9E+09,9E+09,9E+09,9E+09,9E+09]];
    CONST robtarget Target_1220:=[[1062.899929696,366.494489218,584.702492742],[0.045502886,-0.061372268,0.997073261,0.002800813],[0,0,0,0],[9E+09,9E+09,9E+09,9E+09,9E+09,9E+09]];
    CONST robtarget Target_1230:=[[1061.673527845,376.419001221,584.702492742],[0.045502886,-0.061372268,0.997073261,0.002800813],[0,0,0,0],[9E+09,9E+09,9E+09,9E+09,9E+09,9E+09]];
    CONST robtarget Target_1240:=[[1060.447125994,386.343513224,584.702492742],[0.045502886,-0.061372268,0.997073261,0.002800813],[0,0,0,0],[9E+09,9E+09,9E+09,9E+09,9E+09,9E+09]];
    CONST robtarget Target_1250:=[[1059.220724143,396.268025227,584.702492742],[0.045502886,-0.061372268,0.997073261,0.002800813],[0,0,0,0],[9E+09,9E+09,9E+09,9E+09,9E+09,9E+09]];
    CONST robtarget Target_1260:=[[1057.994322292,406.19253723,584.702492742],[0.045502886,-0.061372268,0.997073261,0.002800813],[0,0,0,0],[9E+09,9E+09,9E+09,9E+09,9E+09,9E+09]];
    CONST robtarget Target_1270:=[[1056.767920441,416.117049233,584.702492742],[0.045502886,-0.061372268,0.997073261,0.002800813],[0,0,0,0],[9E+09,9E+09,9E+09,9E+09,9E+09,9E+09]];
    CONST robtarget Target_1280:=[[1055.54151859,426.041561237,584.702492742],[0.045502886,-0.061372268,0.997073261,0.002800813],[0,0,0,0],[9E+09,9E+09,9E+09,9E+09,9E+09,9E+09]];
    CONST robtarget Target_1290:=[[1054.315116739,435.96607324,584.702492742],[0.045502886,-0.061372268,0.997073261,0.002800813],[0,0,0,0],[9E+09,9E+09,9E+09,9E+09,9E+09,9E+09]];
    CONST robtarget Target_1300:=[[1053.088714888,445.890585243,584.702492742],[0.045502886,-0.061372268,0.997073261,0.002800813],[0,0,0,0],[9E+09,9E+09,9E+09,9E+09,9E+09,9E+09]];
    CONST robtarget Target_1310:=[[1051.862313037,455.815097246,584.702492742],[0.045502886,-0.061372268,0.997073261,0.002800813],[0,0,0,0],[9E+09,9E+09,9E+09,9E+09,9E+09,9E+09]];
    CONST robtarget Target_1320:=[[1050.635911186,465.739609249,584.702492742],[0.045502886,-0.061372268,0.997073261,0.002800813],[0,0,0,0],[9E+09,9E+09,9E+09,9E+09,9E+09,9E+09]];
    CONST robtarget Target_1330:=[[1049.409509335,475.664121252,584.702492742],[0.045502886,-0.061372268,0.997073261,0.002800813],[0,0,0,0],[9E+09,9E+09,9E+09,9E+09,9E+09,9E+09]];
    CONST robtarget Target_1340:=[[1048.183107484,485.588633255,584.702492742],[0.045502886,-0.061372268,0.997073261,0.002800813],[0,0,0,0],[9E+09,9E+09,9E+09,9E+09,9E+09,9E+09]];
    CONST robtarget Target_1350:=[[1046.956705633,495.513145258,584.702492742],[0.045502886,-0.061372268,0.997073261,0.002800813],[0,0,0,0],[9E+09,9E+09,9E+09,9E+09,9E+09,9E+09]];
    CONST robtarget Target_1360:=[[1037.073446992,494.29184121,583.791660679],[0.045502886,-0.061372268,0.997073261,0.002800813],[0,0,0,0],[9E+09,9E+09,9E+09,9E+09,9E+09,9E+09]];
    CONST robtarget Target_1370:=[[1027.19018835,493.070537161,582.880828616],[0.045502886,-0.061372268,0.997073261,0.002800813],[0,0,0,0],[9E+09,9E+09,9E+09,9E+09,9E+09,9E+09]];
    CONST robtarget Target_1380:=[[1017.306929709,491.849233112,581.969996552],[0.045502886,-0.061372268,0.997073261,0.002800813],[0,0,0,0],[9E+09,9E+09,9E+09,9E+09,9E+09,9E+09]];
    CONST robtarget Target_1390:=[[1007.423671067,490.627929063,581.059164489],[0.045502886,-0.061372268,0.997073261,0.002800813],[0,0,0,0],[9E+09,9E+09,9E+09,9E+09,9E+09,9E+09]];
    CONST robtarget Target_1400:=[[997.540412426,489.406625014,580.148332426],[0.045502886,-0.061372268,0.997073261,0.002800813],[0,0,0,0],[9E+09,9E+09,9E+09,9E+09,9E+09,9E+09]];
    CONST robtarget Target_1410:=[[987.657153785,488.185320966,579.237500363],[0.045502886,-0.061372268,0.997073261,0.002800813],[0,0,0,0],[9E+09,9E+09,9E+09,9E+09,9E+09,9E+09]];
    CONST robtarget Target_1420:=[[977.773895143,486.964016917,578.3266683],[0.045502886,-0.061372268,0.997073261,0.002800813],[0,0,0,0],[9E+09,9E+09,9E+09,9E+09,9E+09,9E+09]];
    CONST robtarget Target_1430:=[[967.890636502,485.742712868,577.415836236],[0.045502886,-0.061372268,0.997073261,0.002800813],[0,0,0,0],[9E+09,9E+09,9E+09,9E+09,9E+09,9E+09]];
    CONST robtarget Target_1440:=[[958.00737786,484.521408819,576.505004173],[0.045502886,-0.061372268,0.997073261,0.002800813],[0,0,0,0],[9E+09,9E+09,9E+09,9E+09,9E+09,9E+09]];
    CONST robtarget Target_1450:=[[948.124119219,483.300104771,575.59417211],[0.045502886,-0.061372268,0.997073261,0.002800813],[0,0,0,0],[9E+09,9E+09,9E+09,9E+09,9E+09,9E+09]];
    CONST robtarget Target_1460:=[[938.240860578,482.078800722,574.683340047],[0.045502886,-0.061372268,0.997073261,0.002800813],[0,0,0,0],[9E+09,9E+09,9E+09,9E+09,9E+09,9E+09]];
    CONST robtarget Target_1470:=[[928.357601936,480.857496673,573.772507984],[0.045502886,-0.061372268,0.997073261,0.002800813],[0,0,0,0],[9E+09,9E+09,9E+09,9E+09,9E+09,9E+09]];
    CONST robtarget Target_1480:=[[918.474343295,479.636192624,572.861675921],[0.045502886,-0.061372268,0.997073261,0.002800813],[0,0,0,0],[9E+09,9E+09,9E+09,9E+09,9E+09,9E+09]];
    CONST robtarget Target_1490:=[[908.591084653,478.414888575,571.950843857],[0.045502886,-0.061372268,0.997073261,0.002800813],[0,0,0,0],[9E+09,9E+09,9E+09,9E+09,9E+09,9E+09]];
    CONST robtarget Target_1500:=[[898.707826012,477.193584527,571.040011794],[0.045502886,-0.061372268,0.997073261,0.002800813],[0,0,0,0],[9E+09,9E+09,9E+09,9E+09,9E+09,9E+09]];
    CONST robtarget Target_1510:=[[888.824567371,475.972280478,570.129179731],[0.045502886,-0.061372268,0.997073261,0.002800813],[0,0,0,0],[9E+09,9E+09,9E+09,9E+09,9E+09,9E+09]];
    CONST robtarget Target_1520:=[[878.941308729,474.750976429,569.218347668],[0.045502886,-0.061372268,0.997073261,0.002800813],[0,0,0,0],[9E+09,9E+09,9E+09,9E+09,9E+09,9E+09]];
    CONST robtarget Target_1530:=[[869.058050088,473.52967238,568.307515605],[0.045502886,-0.061372268,0.997073261,0.002800813],[0,0,0,0],[9E+09,9E+09,9E+09,9E+09,9E+09,9E+09]];
    CONST robtarget Target_1540:=[[859.174791446,472.308368332,567.396683541],[0.045502886,-0.061372268,0.997073261,0.002800813],[0,0,0,0],[9E+09,9E+09,9E+09,9E+09,9E+09,9E+09]];
    CONST robtarget Target_1550:=[[849.291532805,471.087064283,566.485851478],[0.045502886,-0.061372268,0.997073261,0.002800813],[0,0,0,0],[9E+09,9E+09,9E+09,9E+09,9E+09,9E+09]];
    CONST robtarget Target_1560:=[[839.408274163,469.865760234,565.575019415],[0.045502886,-0.061372268,0.997073261,0.002800813],[0,0,0,0],[9E+09,9E+09,9E+09,9E+09,9E+09,9E+09]];
    CONST robtarget Target_1570:=[[829.525015522,468.644456185,564.664187352],[0.045502886,-0.061372268,0.997073261,0.002800813],[0,0,0,0],[9E+09,9E+09,9E+09,9E+09,9E+09,9E+09]];
    CONST robtarget Target_1580:=[[819.641756881,467.423152136,563.753355289],[0.045502886,-0.061372268,0.997073261,0.002800813],[0,0,0,0],[9E+09,9E+09,9E+09,9E+09,9E+09,9E+09]];
    CONST robtarget Target_1590:=[[809.758498239,466.201848088,562.842523225],[0.045502886,-0.061372268,0.997073261,0.002800813],[0,0,0,0],[9E+09,9E+09,9E+09,9E+09,9E+09,9E+09]];
    CONST robtarget Target_1600:=[[799.875239598,464.980544039,561.931691162],[0.045502886,-0.061372268,0.997073261,0.002800813],[0,0,0,0],[9E+09,9E+09,9E+09,9E+09,9E+09,9E+09]];
    CONST robtarget Target_1610:=[[789.991980956,463.75923999,561.020859099],[0.045502886,-0.061372268,0.997073261,0.002800813],[0,0,0,0],[9E+09,9E+09,9E+09,9E+09,9E+09,9E+09]];
    CONST robtarget Target_1620:=[[780.108722315,462.537935941,560.110027036],[0.045502886,-0.061372268,0.997073261,0.002800813],[0,0,0,0],[9E+09,9E+09,9E+09,9E+09,9E+09,9E+09]];
    CONST robtarget Target_1630:=[[770.225463674,461.316631893,559.199194973],[0.045502886,-0.061372268,0.997073261,0.002800813],[0,0,0,0],[9E+09,9E+09,9E+09,9E+09,9E+09,9E+09]];
    CONST robtarget Target_1640:=[[760.342205032,460.095327844,558.288362909],[0.045502886,-0.061372268,0.997073261,0.002800813],[0,0,0,0],[9E+09,9E+09,9E+09,9E+09,9E+09,9E+09]];
    CONST robtarget Target_1650:=[[750.458946391,458.874023795,557.377530846],[0.045502886,-0.061372268,0.997073261,0.002800813],[0,0,0,0],[9E+09,9E+09,9E+09,9E+09,9E+09,9E+09]];
    CONST robtarget Target_1660:=[[740.575687749,457.652719746,556.466698783],[0.045502886,-0.061372268,0.997073261,0.002800813],[0,0,0,0],[9E+09,9E+09,9E+09,9E+09,9E+09,9E+09]];
    CONST robtarget Target_1670:=[[730.692429108,456.431415697,555.55586672],[0.045502886,-0.061372268,0.997073261,0.002800813],[0,0,0,0],[9E+09,9E+09,9E+09,9E+09,9E+09,9E+09]];
    CONST robtarget Target_1680:=[[720.809170466,455.210111649,554.645034657],[0.045502886,-0.061372268,0.997073261,0.002800813],[0,0,0,0],[9E+09,9E+09,9E+09,9E+09,9E+09,9E+09]];
    CONST robtarget Target_1690:=[[710.925911825,453.9888076,553.734202594],[0.045502886,-0.061372268,0.997073261,0.002800813],[0,0,0,0],[9E+09,9E+09,9E+09,9E+09,9E+09,9E+09]];
    CONST robtarget Target_1700:=[[701.042653184,452.767503551,552.82337053],[0.045502886,-0.061372268,0.997073261,0.002800813],[0,0,0,0],[9E+09,9E+09,9E+09,9E+09,9E+09,9E+09]];
    CONST robtarget Target_1710:=[[691.159394542,451.546199502,551.912538467],[0.045502886,-0.061372268,0.997073261,0.002800813],[0,0,0,0],[9E+09,9E+09,9E+09,9E+09,9E+09,9E+09]];
    CONST robtarget Target_1720:=[[681.276135901,450.324895454,551.001706404],[0.045502886,-0.061372268,0.997073261,0.002800813],[0,0,0,0],[9E+09,9E+09,9E+09,9E+09,9E+09,9E+09]];
    CONST robtarget Target_1730:=[[671.392877259,449.103591405,550.090874341],[0.045502886,-0.061372268,0.997073261,0.002800813],[0,0,0,0],[9E+09,9E+09,9E+09,9E+09,9E+09,9E+09]];
    CONST robtarget Target_1740:=[[661.509618618,447.882287356,549.180042278],[0.045502886,-0.061372268,0.997073261,0.002800813],[0,0,0,0],[9E+09,9E+09,9E+09,9E+09,9E+09,9E+09]];
    CONST robtarget Target_1750:=[[651.626359977,446.660983307,548.269210214],[0.045502886,-0.061372268,0.997073261,0.002800813],[0,0,0,0],[9E+09,9E+09,9E+09,9E+09,9E+09,9E+09]];
    CONST robtarget Target_1760:=[[652.852761828,436.736471304,548.269210214],[0.045502886,-0.061372268,0.997073261,0.002800813],[0,0,0,0],[9E+09,9E+09,9E+09,9E+09,9E+09,9E+09]];
    CONST robtarget Target_1770:=[[654.079163679,426.811959301,548.269210214],[0.045502886,-0.061372268,0.997073261,0.002800813],[0,0,0,0],[9E+09,9E+09,9E+09,9E+09,9E+09,9E+09]];
    CONST robtarget Target_1780:=[[655.305565529,416.887447298,548.269210214],[0.045502886,-0.061372268,0.997073261,0.002800813],[0,0,0,0],[9E+09,9E+09,9E+09,9E+09,9E+09,9E+09]];
    CONST robtarget Target_1790:=[[656.53196738,406.962935295,548.269210214],[0.045502886,-0.061372268,0.997073261,0.002800813],[0,0,0,0],[9E+09,9E+09,9E+09,9E+09,9E+09,9E+09]];
    CONST robtarget Target_1800:=[[657.758369231,397.038423292,548.269210214],[0.045502886,-0.061372268,0.997073261,0.002800813],[0,0,0,0],[9E+09,9E+09,9E+09,9E+09,9E+09,9E+09]];
    CONST robtarget Target_1810:=[[658.984771082,387.113911289,548.269210214],[0.045502886,-0.061372268,0.997073261,0.002800813],[0,0,0,0],[9E+09,9E+09,9E+09,9E+09,9E+09,9E+09]];
    CONST robtarget Target_1820:=[[660.211172933,377.189399285,548.269210214],[0.045502886,-0.061372268,0.997073261,0.002800813],[0,0,0,0],[9E+09,9E+09,9E+09,9E+09,9E+09,9E+09]];
    CONST robtarget Target_1830:=[[661.437574784,367.264887282,548.269210214],[0.045502886,-0.061372268,0.997073261,0.002800813],[0,0,0,0],[9E+09,9E+09,9E+09,9E+09,9E+09,9E+09]];
    CONST robtarget Target_1840:=[[662.663976635,357.340375279,548.269210214],[0.045502886,-0.061372268,0.997073261,0.002800813],[0,0,0,0],[9E+09,9E+09,9E+09,9E+09,9E+09,9E+09]];
    CONST robtarget Target_1850:=[[663.890378486,347.415863276,548.269210214],[0.045502886,-0.061372268,0.997073261,0.002800813],[0,0,0,0],[9E+09,9E+09,9E+09,9E+09,9E+09,9E+09]];
    CONST robtarget Target_1860:=[[665.116780337,337.491351273,548.269210214],[0.045502886,-0.061372268,0.997073261,0.002800813],[0,0,0,0],[9E+09,9E+09,9E+09,9E+09,9E+09,9E+09]];
    CONST robtarget Target_1870:=[[666.343182188,327.56683927,548.269210214],[0.045502886,-0.061372268,0.997073261,0.002800813],[0,0,0,0],[9E+09,9E+09,9E+09,9E+09,9E+09,9E+09]];
    CONST robtarget Target_1880:=[[667.569584039,317.642327267,548.269210214],[0.045502886,-0.061372268,0.997073261,0.002800813],[0,0,0,0],[9E+09,9E+09,9E+09,9E+09,9E+09,9E+09]];
    CONST robtarget Target_1890:=[[668.79598589,307.717815264,548.269210214],[0.045502886,-0.061372268,0.997073261,0.002800813],[0,0,0,0],[9E+09,9E+09,9E+09,9E+09,9E+09,9E+09]];
    CONST robtarget Target_1900:=[[670.022387741,297.793303261,548.269210214],[0.045502886,-0.061372268,0.997073261,0.002800813],[0,0,0,0],[9E+09,9E+09,9E+09,9E+09,9E+09,9E+09]];
    CONST robtarget Target_1910:=[[671.248789592,287.868791257,548.269210214],[0.045502886,-0.061372268,0.997073261,0.002800813],[0,0,0,0],[9E+09,9E+09,9E+09,9E+09,9E+09,9E+09]];
    CONST robtarget Target_1920:=[[672.475191443,277.944279254,548.269210214],[0.045502886,-0.061372268,0.997073261,0.002800813],[0,0,0,0],[9E+09,9E+09,9E+09,9E+09,9E+09,9E+09]];
    CONST robtarget Target_1930:=[[673.701593294,268.019767251,548.269210214],[0.045502886,-0.061372268,0.997073261,0.002800813],[0,0,0,0],[9E+09,9E+09,9E+09,9E+09,9E+09,9E+09]];
    CONST robtarget Target_1940:=[[674.927995145,258.095255248,548.269210214],[0.045502886,-0.061372268,0.997073261,0.002800813],[0,0,0,0],[9E+09,9E+09,9E+09,9E+09,9E+09,9E+09]];
    CONST robtarget Target_1950:=[[676.154396996,248.170743245,548.269210214],[0.045502886,-0.061372268,0.997073261,0.002800813],[0,0,0,0],[9E+09,9E+09,9E+09,9E+09,9E+09,9E+09]];
    CONST robtarget Target_1960:=[[677.380798847,238.246231242,548.269210214],[0.045502886,-0.061372268,0.997073261,0.002800813],[0,0,0,0],[9E+09,9E+09,9E+09,9E+09,9E+09,9E+09]];
    CONST robtarget Target_1970:=[[678.607200698,228.321719239,548.269210214],[0.045502886,-0.061372268,0.997073261,0.002800813],[0,0,0,0],[9E+09,9E+09,9E+09,9E+09,9E+09,9E+09]];
    CONST robtarget Target_1980:=[[679.833602549,218.397207236,548.269210214],[0.045502886,-0.061372268,0.997073261,0.002800813],[0,0,0,0],[9E+09,9E+09,9E+09,9E+09,9E+09,9E+09]];
    CONST robtarget Target_1990:=[[681.0600044,208.472695233,548.269210214],[0.045502886,-0.061372268,0.997073261,0.002800813],[0,0,0,0],[9E+09,9E+09,9E+09,9E+09,9E+09,9E+09]];
    CONST robtarget Target_2000:=[[682.286406251,198.548183229,548.269210214],[0.045502886,-0.061372268,0.997073261,0.002800813],[0,0,0,0],[9E+09,9E+09,9E+09,9E+09,9E+09,9E+09]];
    CONST robtarget Target_2010:=[[683.512808102,188.623671226,548.269210214],[0.045502886,-0.061372268,0.997073261,0.002800813],[0,0,0,0],[9E+09,9E+09,9E+09,9E+09,9E+09,9E+09]];
    CONST robtarget Target_2020:=[[684.739209953,178.699159223,548.269210214],[0.045502886,-0.061372268,0.997073261,0.002800813],[0,0,0,0],[9E+09,9E+09,9E+09,9E+09,9E+09,9E+09]];
    CONST robtarget Target_2030:=[[685.965611804,168.77464722,548.269210214],[0.045502886,-0.061372268,0.997073261,0.002800813],[0,0,0,0],[9E+09,9E+09,9E+09,9E+09,9E+09,9E+09]];
    CONST robtarget Target_2040:=[[687.192013655,158.850135217,548.269210214],[0.045502886,-0.061372268,0.997073261,0.002800813],[0,0,0,0],[9E+09,9E+09,9E+09,9E+09,9E+09,9E+09]];
    CONST robtarget Target_2050:=[[688.418415506,148.925623214,548.269210214],[0.045502886,-0.061372268,0.997073261,0.002800813],[0,0,0,0],[9E+09,9E+09,9E+09,9E+09,9E+09,9E+09]];
    CONST robtarget Target_2060:=[[698.301674147,150.146927263,549.180042278],[0.045502886,-0.061372268,0.997073261,0.002800813],[0,0,0,0],[9E+09,9E+09,9E+09,9E+09,9E+09,9E+09]];
    CONST robtarget Target_2070:=[[708.184932789,151.368231311,550.090874341],[0.045502886,-0.061372268,0.997073261,0.002800813],[0,0,0,0],[9E+09,9E+09,9E+09,9E+09,9E+09,9E+09]];
    CONST robtarget Target_2080:=[[718.06819143,152.58953536,551.001706404],[0.045502886,-0.061372268,0.997073261,0.002800813],[0,0,0,0],[9E+09,9E+09,9E+09,9E+09,9E+09,9E+09]];
    CONST robtarget Target_2090:=[[727.951450072,153.810839409,551.912538467],[0.045502886,-0.061372268,0.997073261,0.002800813],[0,0,0,0],[9E+09,9E+09,9E+09,9E+09,9E+09,9E+09]];
    CONST robtarget Target_2100:=[[737.834708713,155.032143458,552.82337053],[0.045502886,-0.061372268,0.997073261,0.002800813],[0,0,0,0],[9E+09,9E+09,9E+09,9E+09,9E+09,9E+09]];
    CONST robtarget Target_2110:=[[747.717967354,156.253447507,553.734202594],[0.045502886,-0.061372268,0.997073261,0.002800813],[0,0,0,0],[9E+09,9E+09,9E+09,9E+09,9E+09,9E+09]];
    CONST robtarget Target_2120:=[[757.601225996,157.474751555,554.645034657],[0.045502886,-0.061372268,0.997073261,0.002800813],[0,0,0,0],[9E+09,9E+09,9E+09,9E+09,9E+09,9E+09]];
    CONST robtarget Target_2130:=[[767.484484637,158.696055604,555.55586672],[0.045502886,-0.061372268,0.997073261,0.002800813],[0,0,0,0],[9E+09,9E+09,9E+09,9E+09,9E+09,9E+09]];
    CONST robtarget Target_2140:=[[777.367743279,159.917359653,556.466698783],[0.045502886,-0.061372268,0.997073261,0.002800813],[0,0,0,0],[9E+09,9E+09,9E+09,9E+09,9E+09,9E+09]];
    CONST robtarget Target_2150:=[[787.25100192,161.138663702,557.377530846],[0.045502886,-0.061372268,0.997073261,0.002800813],[0,0,0,0],[9E+09,9E+09,9E+09,9E+09,9E+09,9E+09]];
    CONST robtarget Target_2160:=[[797.134260562,162.35996775,558.288362909],[0.045502886,-0.061372268,0.997073261,0.002800813],[0,0,0,0],[9E+09,9E+09,9E+09,9E+09,9E+09,9E+09]];
    CONST robtarget Target_2170:=[[807.017519203,163.581271799,559.199194973],[0.045502886,-0.061372268,0.997073261,0.002800813],[0,0,0,0],[9E+09,9E+09,9E+09,9E+09,9E+09,9E+09]];
    CONST robtarget Target_2180:=[[816.900777844,164.802575848,560.110027036],[0.045502886,-0.061372268,0.997073261,0.002800813],[0,0,0,0],[9E+09,9E+09,9E+09,9E+09,9E+09,9E+09]];
    CONST robtarget Target_2190:=[[826.784036486,166.023879897,561.020859099],[0.045502886,-0.061372268,0.997073261,0.002800813],[0,0,0,0],[9E+09,9E+09,9E+09,9E+09,9E+09,9E+09]];
    CONST robtarget Target_2200:=[[836.667295127,167.245183946,561.931691162],[0.045502886,-0.061372268,0.997073261,0.002800813],[0,0,0,0],[9E+09,9E+09,9E+09,9E+09,9E+09,9E+09]];
    CONST robtarget Target_2210:=[[846.550553769,168.466487994,562.842523225],[0.045502886,-0.061372268,0.997073261,0.002800813],[0,0,0,0],[9E+09,9E+09,9E+09,9E+09,9E+09,9E+09]];
    CONST robtarget Target_2220:=[[856.43381241,169.687792043,563.753355289],[0.045502886,-0.061372268,0.997073261,0.002800813],[0,0,0,0],[9E+09,9E+09,9E+09,9E+09,9E+09,9E+09]];
    CONST robtarget Target_2230:=[[866.317071051,170.909096092,564.664187352],[0.045502886,-0.061372268,0.997073261,0.002800813],[0,0,0,0],[9E+09,9E+09,9E+09,9E+09,9E+09,9E+09]];
    CONST robtarget Target_2240:=[[876.200329693,172.130400141,565.575019415],[0.045502886,-0.061372268,0.997073261,0.002800813],[0,0,0,0],[9E+09,9E+09,9E+09,9E+09,9E+09,9E+09]];
    CONST robtarget Target_2250:=[[886.083588334,173.351704189,566.485851478],[0.045502886,-0.061372268,0.997073261,0.002800813],[0,0,0,0],[9E+09,9E+09,9E+09,9E+09,9E+09,9E+09]];
    CONST robtarget Target_2260:=[[895.966846976,174.573008238,567.396683541],[0.045502886,-0.061372268,0.997073261,0.002800813],[0,0,0,0],[9E+09,9E+09,9E+09,9E+09,9E+09,9E+09]];
    CONST robtarget Target_2270:=[[905.850105617,175.794312287,568.307515605],[0.045502886,-0.061372268,0.997073261,0.002800813],[0,0,0,0],[9E+09,9E+09,9E+09,9E+09,9E+09,9E+09]];
    CONST robtarget Target_2280:=[[915.733364258,177.015616336,569.218347668],[0.045502886,-0.061372268,0.997073261,0.002800813],[0,0,0,0],[9E+09,9E+09,9E+09,9E+09,9E+09,9E+09]];
    CONST robtarget Target_2290:=[[925.6166229,178.236920385,570.129179731],[0.045502886,-0.061372268,0.997073261,0.002800813],[0,0,0,0],[9E+09,9E+09,9E+09,9E+09,9E+09,9E+09]];
    CONST robtarget Target_2300:=[[935.499881541,179.458224433,571.040011794],[0.045502886,-0.061372268,0.997073261,0.002800813],[0,0,0,0],[9E+09,9E+09,9E+09,9E+09,9E+09,9E+09]];
    CONST robtarget Target_2310:=[[945.383140183,180.679528482,571.950843857],[0.045502886,-0.061372268,0.997073261,0.002800813],[0,0,0,0],[9E+09,9E+09,9E+09,9E+09,9E+09,9E+09]];
    CONST robtarget Target_2320:=[[955.266398824,181.900832531,572.861675921],[0.045502886,-0.061372268,0.997073261,0.002800813],[0,0,0,0],[9E+09,9E+09,9E+09,9E+09,9E+09,9E+09]];
    CONST robtarget Target_2330:=[[965.149657466,183.12213658,573.772507984],[0.045502886,-0.061372268,0.997073261,0.002800813],[0,0,0,0],[9E+09,9E+09,9E+09,9E+09,9E+09,9E+09]];
    CONST robtarget Target_2340:=[[975.032916107,184.343440628,574.683340047],[0.045502886,-0.061372268,0.997073261,0.002800813],[0,0,0,0],[9E+09,9E+09,9E+09,9E+09,9E+09,9E+09]];
    CONST robtarget Target_2350:=[[984.916174748,185.564744677,575.59417211],[0.045502886,-0.061372268,0.997073261,0.002800813],[0,0,0,0],[9E+09,9E+09,9E+09,9E+09,9E+09,9E+09]];
    CONST robtarget Target_2360:=[[994.79943339,186.786048726,576.505004173],[0.045502886,-0.061372268,0.997073261,0.002800813],[0,0,0,0],[9E+09,9E+09,9E+09,9E+09,9E+09,9E+09]];
    CONST robtarget Target_2370:=[[1004.682692031,188.007352775,577.415836236],[0.045502886,-0.061372268,0.997073261,0.002800813],[0,0,0,0],[9E+09,9E+09,9E+09,9E+09,9E+09,9E+09]];
    CONST robtarget Target_2380:=[[1014.565950673,189.228656823,578.3266683],[0.045502886,-0.061372268,0.997073261,0.002800813],[0,0,0,0],[9E+09,9E+09,9E+09,9E+09,9E+09,9E+09]];
    CONST robtarget Target_2390:=[[1024.449209314,190.449960872,579.237500363],[0.045502886,-0.061372268,0.997073261,0.002800813],[0,0,0,0],[9E+09,9E+09,9E+09,9E+09,9E+09,9E+09]];
    CONST robtarget Target_2400:=[[1034.332467955,191.671264921,580.148332426],[0.045502886,-0.061372268,0.997073261,0.002800813],[0,0,0,0],[9E+09,9E+09,9E+09,9E+09,9E+09,9E+09]];
    CONST robtarget Target_2410:=[[1044.215726597,192.89256897,581.059164489],[0.045502886,-0.061372268,0.997073261,0.002800813],[0,0,0,0],[9E+09,9E+09,9E+09,9E+09,9E+09,9E+09]];
    CONST robtarget Target_2420:=[[1054.098985238,194.113873019,581.969996552],[0.045502886,-0.061372268,0.997073261,0.002800813],[0,0,0,0],[9E+09,9E+09,9E+09,9E+09,9E+09,9E+09]];
    CONST robtarget Target_2430:=[[1063.98224388,195.335177067,582.880828616],[0.045502886,-0.061372268,0.997073261,0.002800813],[0,0,0,0],[9E+09,9E+09,9E+09,9E+09,9E+09,9E+09]];
    CONST robtarget Target_2440:=[[1073.865502521,196.556481116,583.791660679],[0.045502886,-0.061372268,0.997073261,0.002800813],[0,0,0,0],[9E+09,9E+09,9E+09,9E+09,9E+09,9E+09]];
! Module:  Module1
    !
    ! Description:
    !   <Insert description here>
    !
    ! Author: Administrator
    !
    ! Version: 1.0
    !
    !***********************************************************


    !***********************************************************
    !
    ! Procedure main
    !
    !   This is the entry point of your program
    !
    !***********************************************************


    PROC main()

       VAR num sum;
       VAR bool bExit:=FALSE;

       WHILE NOT bExit DO
            Incr sum;
            IF sum = 10 THEN
                TPWrite "Sum :" \Num:= sum;
                bExit:=TRUE;
                ! ----------  Exit while loop and continue command
            ENDIF
            Path_10;
            WaitTime 3;
            Path_20;
            WaitTime 3;
       ENDWHILE


    ENDPROC


ENDMODULE

--- Backups/IRB_1520ID_4kg_1.50m/RAPID/TASK1/SYSMOD/LINKEDM.sys ---
%%%
  VERSION:1
  LANGUAGE:ENGLISH
%%%

MODULE LINKEDM (SYSMODULE)

! FOLLOWER
!     Name of electronically linked follower axis used by operator at teach pendent.
      PERS string l_f_axis_name{5}       :=  ["",  "", "", "", ""];

!     Name of the mechanical unit for follower axis.
      PERS string l_f_mecunt_n{5}  :=  ["", "", "", "", ""];

!     Linked follower axis number in the mechanical unit (first axis in mech. unit is number 1).
      PERS num l_f_axis_no{5}      :=  [0,          0,   0,  0,  0];

! MASTER
!     Name of the mechanical unit for linked master axis.
      PERS string l_m_mecunt_n{5} :=  ["", "", "", "", ""];

!     Linked master axis number in the mechanical unit (first axis in mech. unit is number 1).
!     See axis number table in documentation for different master mechanical units.
      PERS num l_m_axis_no{5}     :=  [0,  0,  0,  0,  0];

! POSITION OFFSET
!     The increase of the allowed offset position between the master and follower
!     positions, used when starting AUTO mode. As soon as the offset is decreased
!     the old configurated parameter is used.
!     Example: 3 => the configurated value of allowed offset is increased 3 times.
      PERS num offset_ratio{5}       :=  [10,  10,   10,  10,  10];

! SPEED RATIO
!     Speed_ratio used in AUTO and JOG modes [ very_slow   slow    normal    fast]
!     Value 1 = max allowed manual speed.
      CONST num speed_ratio {20}      := [0.01, 0.01, 0.01, 0.01, 0.01,
                                          0.05, 0.05, 0.05, 0.05, 0.05,
                                          0.20, 0.20, 0.20, 0.20, 0.20,
                                          1.00, 1.00, 1.00, 1.00, 1.00];

! STEP SIZE
!     Displacement position used in JOG mode for each activation of positive or
!     negative movement.                  [very_short    short   normal   long]
!     Unit degees or meter.
      CONST num displacement {20}     := [0.001, 0.001, 0.001, 0.001, 0.001,
                                          0.005, 0.005, 0.005, 0.005, 0.005,
                                          0.020, 0.020, 0.020, 0.020, 0.020,
                                          0.100, 0.100, 0.100, 0.100, 0.100];


!-------------------------------------------------------------
 PROC Linked_m ()
      Linked_m_exe ;
 ENDPROC
ENDMODULE
